# B&R Automation Studio project spro4_pendulum
Automation Studio 4.12.6.106; technology packages: Acp10Arnc0 5.31.0

## Configuration Config1

CPU X20CP1382, AutomationRuntime H4.83, Build 4.1.2, Vc V4.73.2

### Task classes (Cpu.sw)
```
Cyclic#1 (cycle 2000 us):
  Program <- Program.prg
Binaries: udbdef, FWRules, TCData, sysconf, Role, User, iomap, ashwd, asfw, arconfig, ashwac
Libraries: standard, runtime, astime, asieccon, AsMath
```

### Hardware
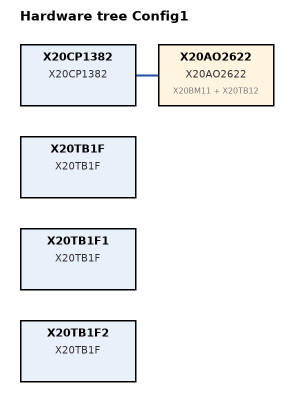
```
X20AO2622 : X20AO2622 v1.3.0.0  [SS1 -> X20TB12.SS; SL -> X20BM11.SL1]
X20BM11 : X20BM11 v1.1.0.0  [X2X1 -> X20CP1382.IF6]
X20CP1382 : X20CP1382 v1.15.0.0  [X1 -> X1.SL; X2 -> X2.SL; X3 -> X3.SL]
  Module X1 (Type=X1, Virtual=true, Version=1.15.0.0)
    Connection (Connector=SS1, TargetModule=X20TB1F, TargetConnector=SS)
    Connection (Connector=SL, TargetModule=X20CP1382, TargetConnector=X1)
  Module X2 (Type=X2, Virtual=true, Version=1.15.0.0)
    Connection (Connector=SS1, TargetModule=X20TB1F1, TargetConnector=SS)
    Connection (Connector=SL, TargetModule=X20CP1382, TargetConnector=X2)
    X2CounterFunction = AB
    X2CounterTimeInfo = 32Bit
  Module X3 (Type=X3, Virtual=true, Version=1.15.0.0)
    Connection (Connector=SS1, TargetModule=X20TB1F2, TargetConnector=SS)
    Connection (Connector=SL, TargetModule=X20CP1382, TargetConnector=X3)
  Connector IF2:
    ActivateDevice = 1
    Mode = Manual
    InternetAddress = 192.168.8.101
    SubnetMask = 255.255.255.0
    InaNodeNumber = 0
  ConfigurationID = spro4_pendulum_Config1
  SystemTick = 1000
  Cyclic1Duration = 2000
X20TB12 : X20TB12 v1.0.0.0
X20TB1F : X20TB1F v1.0.0.0
X20TB1F1 : X20TB1F v1.0.0.0
X20TB1F2 : X20TB1F v1.0.0.0
```

### Acp10cfg.ncc - X20CP1382/Motion/Acp10cfg.ncc
```
NcConfiguration (Version=5.31.0, NcSwId=Acp10)
  ACP10CF1_typ:
    cnt_nettrc_rec_drive = 150
    bufsize_trace_upload = 1200
    tc_nc_man_task = Cyclic #1
    glob_pv_as_ncobject = Yes
    ncsys_dl_broadcast = Yes
    ncsys_dl_acp_reset = Yes
    safemc_log_err_to_ax = Yes
    network_init:
      ncsw_init_execute = Yes
      automatic_execute = No
      node_nr_warning = Yes
      net_err_before_ncact = Yes
    nettrc:
      enter_parsecrec = Yes
      enter_ncaction = Yes
      save_ring_startidx = No
    cam_prof_download:
      cam_dat_dl_parallel = No
      tc_cam_dl_parallel = Task class for NC Manager task
```

## Logical view

Binary libraries used (declarations not repeated): operator, runtime, astime, AsIecCon, standard, AsMath, Acp10par 5.31.0

### Global.var
```iecst
VAR
	Q_reset_LED : BOOL;
	SI_estop_B : BOOL;
	SI_estop_A : BOOL;
	I_drive_active : BOOL;
	I_drive_no_fault : BOOL;
	I_endstop_negative : BOOL;
	I_endstop_positive : BOOL;
	I_pos_cart : DINT;
	I_pos_pendulum : DINT;
	Q_drive_enable : BOOL;
	Q_drive_faultreset : BOOL;
	Q_drive_operating_mode : BOOL;
	Q_vel_cart : INT;
	SI_reset_btn : BOOL;
	reset_cart_position : BOOL;
	reset_pendulum_position : BOOL;
END_VAR
```

### Program Logical/Program (IEC)

#### Main.st - Init, cyclic, exit code
```iecst
PROGRAM _INIT // Alt her bruges, må gerne få refactor men ikke ændre funktionalitet

	Q_vel_cart := 0;
	length := 0;
	I_pos_pendulum;
	reset_pendulum_position;
	I_pos_cart;
	reset_cart_position;
	systemState := idle;
	speed := -2000;

	scale := 1310;

END_PROGRAM

PROGRAM _CYCLIC

	// Handle EStop
	IF(SI_estop_A AND SI_estop_B) THEN
		Q_drive_enable := TRUE;
	ELSE
		Q_drive_enable  := FALSE;
		Q_reset_LED := FALSE;
	END_IF

	// Handle Reset Btn
	IF(SI_reset_btn) THEN
		Q_drive_faultreset := NOT Q_drive_faultreset;
	ELSIF I_drive_no_fault THEN
		Q_reset_LED := TRUE;
	ELSE
		led_ton(IN:=NOT led_ton.Q, PT := T#200ms);
		IF(led_ton.Q) THEN
			Q_reset_LED := NOT Q_reset_LED;
		END_IF
	END_IF

	CASE systemState OF // Main state machine
		idle: // Bruges
			resetTimer.IN := FALSE;
			counter := 0;
			Q_vel_cart := 0;
			reset_pendulum_position := FALSE;
			reset_cart_position := FALSE;
			Q_drive_faultreset := NOT Q_drive_faultreset;

			e_prev := 0;
			Fd_prev := 0;
			e_sum := 0;

		reset: // Bruges
			IF NOT I_endstop_positive THEN
				Q_vel_cart := 0;
			ELSE
				Q_vel_cart := 4000;
			END_IF

			resetTimer.IN := (Q_vel_cart = 0); // Timer counts as long as vel is 0
			resetTimer.PT := T#1s; // Timer set to 1 second
			resetTimer();

			IF resetTimer.Q THEN
				reset_pendulum_position := TRUE;
				reset_cart_position := TRUE;

				systemState := idle;
			END_IF

			Q_drive_faultreset := NOT Q_drive_faultreset;

		manual: // Bruges ikke, var tænkt til kontrol med piletaster el.lign.
			IF NOT I_endstop_negative THEN
				systemState := idle;
			END_IF
			Q_vel_cart := -4000;
			Q_drive_faultreset := NOT Q_drive_faultreset;

		swing: // Bruges ikke, tænkt til "swing-up" sequence.
			Q_vel_cart := speed;
			counter := counter + 1;
			IF (counter = 9) THEN
				pos_start := I_pos_cart;
				resetTimer.IN := TRUE;
				resetTimer.PT := T#5s;
			END_IF

			resetTimer();

			IF resetTimer.Q THEN
				pos_end := I_pos_cart;
				systemState := idle;
			END_IF

			IF NOT I_endstop_negative THEN
				systemState := idle;
			END_IF

		controller: // Tidlig test controller, bør gemmes
			IF (I_pos_pendulum > 1700 AND I_pos_pendulum < 2350) THEN
				Q_vel_cart := speed * (DINT_TO_INT(I_pos_pendulum) - 2048);
			ELSE
				Q_vel_cart := 0;
			END_IF
			IF (Q_vel_cart > 10000) THEN
				Q_vel_cart := 10000;
			ELSIF (Q_vel_cart < -10000) THEN
				Q_vel_cart := -10000;
			END_IF
			IF NOT I_endstop_positive OR NOT I_endstop_negative THEN
				Q_vel_cart := 0;
			END_IF

		PDcontroller: // MAIN PID CONTROLLER - NO TOUCH!
			// Cart (outer loop)
			Kp_cart := -0.00234 * 50;
			Ki_cart := 0;
			Kd_cart := -0.00468 * 50;
			Tf_cart := 0.01;
			Ts_cart := 0.002;

			pos_ref := 190000;
			pos := I_pos_cart;

			e_cart := (pos_ref - pos) / 243500;

			e_sum_cart := e_sum_cart + (e_cart * Ts_cart);

			IF e_sum_cart > 100.0 THEN
				e_sum_cart := 100.0;
			ELSIF e_sum_cart < -100.0 THEN
				e_sum_cart := -100.0;
			END_IF

			Fd_cart := (Tf_cart / (Tf_cart + Ts_cart)) * Fd_prev_cart + (Kd_cart / (Tf_cart + Ts_cart)) * (e_cart - e_prev_cart);

			F_cart := Kp_cart * e_cart + Ki_cart * e_sum_cart + Fd_cart;

			e_prev_cart := e_cart;
			Fd_prev_cart := Fd_cart;

			// Pendulum (inner loop)
			Kp := 14.23031;
			Ki := 63.24582;
			Kd := 0.79057;
			Tf := 0.01;
			Ts := 0.002;

			theta_ref := -F_cart;
			theta := (I_pos_pendulum - 2048) * ((2 * amPI) / 4096);

			e := theta_ref - theta;

			e_sum := e_sum + (e * Ts);

			IF e_sum > 100.0 THEN
				e_sum := 100.0;
			ELSIF e_sum < -100.0 THEN
				e_sum := -100.0;
			END_IF

			Fd := (Tf / (Tf + Ts)) * Fd_prev + (Kd / (Tf + Ts)) * (e - e_prev);

			F := Kp * e + Ki * e_sum + Fd;

			e_prev := e;
			Fd_prev := Fd;

			IF (I_pos_pendulum > 1550 AND I_pos_pendulum < 2550) THEN
				Q_vel_cart := REAL_TO_INT(F * scale);
			ELSE
				Q_vel_cart := 0;
				systemState := idle;
			END_IF
			IF (Q_vel_cart > 7500) THEN
				Q_vel_cart := 7500;
			ELSIF (Q_vel_cart < -7500) THEN
				Q_vel_cart := -7500;
			END_IF
			IF NOT I_endstop_positive OR NOT I_endstop_negative THEN
				Q_vel_cart := 0;
				systemState := idle;
			END_IF

			IF (I_pos_cart > 330000 OR I_pos_cart < 50000) THEN
				Q_vel_cart := 0;
				systemState := idle;
			END_IF

			IF Q_vel_cart < 0 THEN
				Q_vel_cart := Q_vel_cart - 1700;
			ELSIF Q_vel_cart > 0 THEN
				Q_vel_cart := Q_vel_cart + 1700;
			END_IF

		center: // Bruges til at bevæge til midten af båndet
			Q_vel_cart := -4000;
			IF (I_pos_cart > 190000) THEN
				systemState := idle;
			END_IF

		Preset: // Bruges til reset af pendul encoder
			reset_pendulum_position := TRUE;
			systemState := idle;

	END_CASE

END_PROGRAM

PROGRAM _EXIT

END_PROGRAM
```

#### Types.typ - Local data types
```iecst
TYPE
	direction :
		(
		cart_stop,
		cart_right,
		cart_left
		);
	system_State :
		(
		controller,
		manual,
		swing,
		reset,
		idle,
		Preset,
		center,
		PDcontroller
		);
END_TYPE
```

#### Variables.var - Local variables
```iecst
VAR
	DIR : direction;
	length : DINT;
	led_ton : TON;
	systemState : system_State := idle;
	resetTimer : TON;
	counter : REAL;
	pos_start : DINT;
	pos_end : DINT;
	speed : INT;
	Ki : REAL;
	Kd : REAL;
	theta : REAL;
	theta_ref : REAL;
	Fd_prev : REAL;
	e_prev : REAL;
	Ts : REAL;
	Tf : REAL;
	Kp : REAL;
	Fd : REAL;
	e : REAL;
	F : REAL;
	scale : INT;
	e_sum : REAL;
	Ki_cart : REAL;
	Kd_cart : REAL;
	pos : REAL;
	pos_ref : REAL;
	Fd_prev_cart : REAL;
	e_prev_cart : REAL;
	Ts_cart : REAL;
	Tf_cart : REAL;
	Kp_cart : REAL;
	Fd_cart : REAL;
	e_cart : REAL;
	F_cart : REAL;
	e_sum_cart : REAL;
END_VAR
```

#### Variables1.var
```iecst
VAR
	alpha : REAL := 0.01;
	K1 : REAL;
	K2 : REAL;
	K3 : REAL;
	K4 : REAL;
	K5 : REAL;
	filt_x_dot : REAL;
	filt_theta_dot : REAL;
	Kd_pen : REAL;
	Ki_pen : REAL;
	Kp_pen : REAL;
	Ki_cart : REAL;
	Kd_cart : REAL;
	Kp_cart : REAL;
	error_x : REAL;
	error_theta : REAL;
	error_x_old : REAL;
	error_theta_old : REAL;
	u_cart : REAL;
	u_i_cart : REAL;
	u_d_cart : REAL;
	u_d_old_cart : REAL;
	u_i_pen : REAL;
	u_d_pen : REAL;
	u_d_old_pen : REAL;
END_VAR
```

#### Variables2.var
```iecst
VAR
	m_p : REAL := 0.084;
	g : REAL := 9.82;
	l : REAL := 0.175;
	I_p : REAL := 0.002572;
	energy_gain : REAL := 15;
	energy : REAL;
	error_energy : REAL;
	theta_cos : REAL;
	direction : REAL;
END_VAR
```
